ABB RobotStudio station: Yummi-Pick-and-Place.rsstn

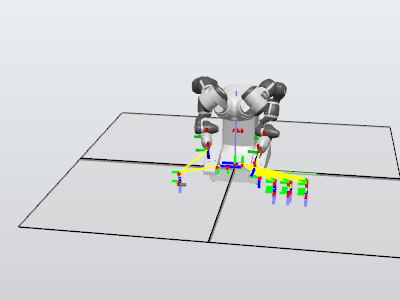
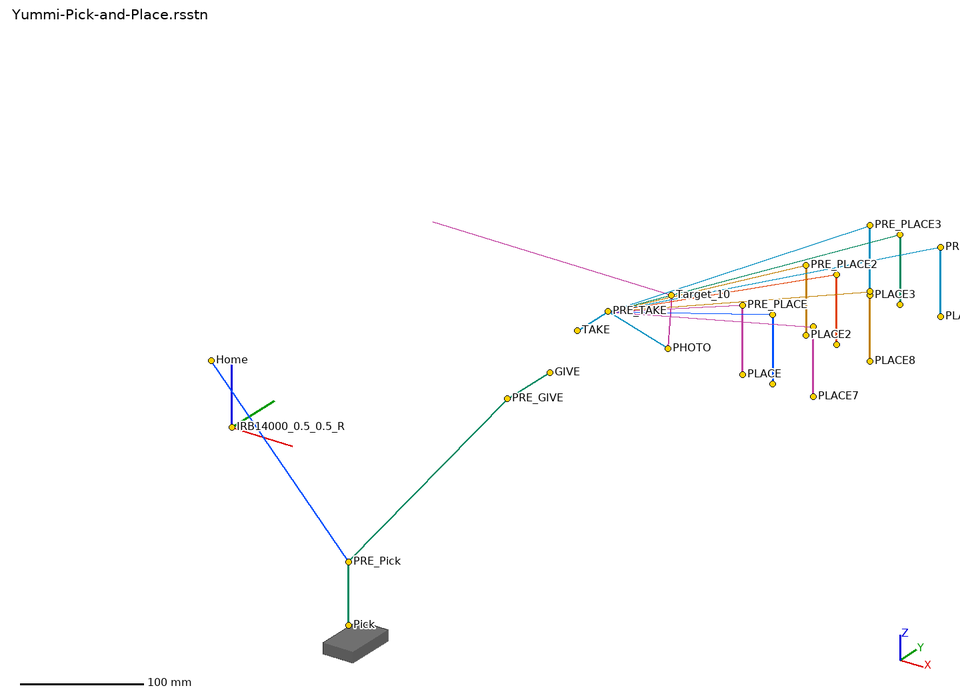
[picture v1: parts stored in the station drawn from their meshes, with robot base, taught points and paths (robot models come from the ABB library and are not in the file)]
Station Yummi5 (saved by RobotStudio 24.3.10958.1)
Controller Controller12
  mechanical unit ROB_R: IRB14000_0.5_0.5_R, 6 joints, base frame (0, 0, 0) mm
  mechanical unit ROB_R_7: IRB14000_0.5_0.5_R, 1 joints, base frame (0, 0, 0) mm
  mechanical unit ROB_L: IRB14000_0.5_0.5_L, 6 joints, base frame (0, 0, 0) mm
  mechanical unit ROB_L_7: IRB14000_0.5_0.5_L, 1 joints, base frame (0, 0, 0) mm
Layout (positions relative to the parent item):
  - IRB14000_0.5_0.5 [mechanism, from %ABB.RobotStudio.Models.IRB14000%\IRB14000_0.5_0.5__02.rslib] at (0, 0, 0) mm
  - IRB14000_0.5_0.5_R [mechanism, from %ABB.RobotStudio.Models.IRB14000%\IRB14000_0.5_0.5__02.rslib] at (0, 0, 0) mm; joint values [1.3686, -2.3546, -0.9667, 0.4669, -1.2245, 1.4931, 2.9439] (rad or m)
  - IRB14000_0.5_0.5_L [mechanism, from %ABB.RobotStudio.Models.IRB14000%\IRB14000_0.5_0.5__02.rslib] at (0, 0, 0) mm; joint values [-1.4023, -1.9659, 0.2989, 0.1537, 2.388, 1.6864, -2.7781] (rad or m)
  - Smart_Gripper_Servo_Fingers [mechanism] at (-9.58, -182.61, 198.63) mm, rotated rx 179.34 ry -63.63 rz 15.45 deg; joint values [0.02] (rad or m)
      TCP Servo at (0, 0, 114.2) mm
      links: HandBase, DownFinger, UpFinger, VacuumOne, VacuumTwo
  - Smart_Gripper_Servo_Fingers_2 [mechanism] at (-9.58, 182.61, 198.63) mm, rotated rx -179.34 ry -63.63 rz -15.45 deg; joint values [0.02] (rad or m)
      TCP Servo at (0, 0, 114.2) mm
      links: HandBase, DownFinger, UpFinger, VacuumOne, VacuumTwo
  - Part_2 [part] at (100, 0, 0) mm, size 30 x 50 x 10 mm
  - Part_3 [part], size 30 x 50 x 10 mm
  - Part_4 [part], size 30 x 50 x 10 mm
  - Part_5 [part], size 30 x 50 x 10 mm
  - Part_6 [part], size 30 x 50 x 10 mm
  - Part_7 [part], size 30 x 50 x 10 mm
  - Part_8 [part], size 30 x 50 x 10 mm
  - Part_9 [part], size 30 x 50 x 10 mm
  - Part_10 [part], size 30 x 50 x 10 mm
Attachment: Smart_Gripper_Servo_Fingers is attached to IRB14000_0.5_0.5_R / Link7
Attachment: Smart_Gripper_Servo_Fingers_2 is attached to IRB14000_0.5_0.5_L / Link7
EventTableEntry 3683: Group=, Trigger=GripperR 3684, Actions=[EventTableActionMechanicalPose 4791, EventTableActionAttach 4792], Comment=, ActivationMode=2, Cyclic=false
EventTableTriggerIO 3684: IOValue=[1], IRC5Controller=? -1, Operator=0, SignalSource=Controller12 1195
EventTableTriggerIO 3686: IOValue=[0], IRC5Controller=? -1, Operator=0, SignalSource=Controller12 1195
EventTableTriggerIO 3687: IOValue=[1], IRC5Controller=? -1, Operator=0, SignalSource=Controller12 1195
EventTableTriggerIO 3688: IOValue=[0], IRC5Controller=? -1, Operator=0, SignalSource=Controller12 1195
EventTableTriggerIO 3689: IOValue=[1], IRC5Controller=? -1, Operator=0, SignalSource=Controller12 1195
EventTableTriggerIO 3690: IOValue=[0], IRC5Controller=? -1, Operator=0, SignalSource=Controller12 1195
EventTableTriggerIO 3691: IOValue=[1], IRC5Controller=? -1, Operator=0, SignalSource=Controller12 1195
EventTableTriggerIO 3692: IOValue=[0], IRC5Controller=? -1, Operator=0, SignalSource=Controller12 1195
EventTableTriggerIO 3693: IOValue=[1], IRC5Controller=? -1, Operator=0, SignalSource=Controller12 1195
EventTableTriggerIO 3694: IOValue=[0], IRC5Controller=? -1, Operator=0, SignalSource=Controller12 1195
EventTableEntry 3695: Group=, Trigger=GripperR 3686, Actions=[EventTableActionMechanicalPose 3696, EventTableActionDetach 4527], Comment=, ActivationMode=2, Cyclic=false
EventTableActionMechanicalPose 3696: VirtualSignal=, Mechanism=Smart_Gripper_Servo_Fingers 3661, ToPoseName=Pose2, VirtualSignalValue=[1]
EventTableTriggerIO 3853: IOValue=[1], IRC5Controller=? -1, Operator=0, SignalSource=Controller12 1195
EventTableTriggerIO 3854: IOValue=[0], IRC5Controller=? -1, Operator=0, SignalSource=Controller12 1195
EventTableTriggerIO 3855: IOValue=[1], IRC5Controller=? -1, Operator=0, SignalSource=Controller12 1195
EventTableTriggerIO 3856: IOValue=[0], IRC5Controller=? -1, Operator=0, SignalSource=Controller12 1195
EventTableEntry 4149: Group=, Trigger=GripperL 4150, Actions=[EventTableActionMechanicalPose 4151, EventTableActionAttach 4528], Comment=, ActivationMode=2, Cyclic=false
EventTableTriggerIO 4150: IOValue=[1], IRC5Controller=? -1, Operator=0, SignalSource=Controller12 1195
EventTableActionMechanicalPose 4151: VirtualSignal=, Mechanism=Smart_Gripper_Servo_Fingers_2 3668, ToPoseName=Pose1, VirtualSignalValue=[1]
EventTableTriggerIO 4152: IOValue=[0], IRC5Controller=? -1, Operator=0, SignalSource=Controller12 1195
EventTableEntry 4153: Group=, Trigger=GripperL 4152, Actions=[EventTableActionMechanicalPose 4154, EventTableActionDetach 4529], Comment=, ActivationMode=2, Cyclic=false
EventTableActionMechanicalPose 4154: VirtualSignal=, Mechanism=Smart_Gripper_Servo_Fingers_2 3668, ToPoseName=Pose2, VirtualSignalValue=[1]
EventTableTriggerIO 4291: IOValue=[1], IRC5Controller=? -1, Operator=0, SignalSource=Controller12 1195
EventTableTriggerIO 4292: IOValue=[0], IRC5Controller=? -1, Operator=0, SignalSource=Controller12 1195
EventTableTriggerIO 4293: IOValue=[1], IRC5Controller=? -1, Operator=0, SignalSource=Controller12 1195
EventTableTriggerIO 4294: IOValue=[0], IRC5Controller=? -1, Operator=0, SignalSource=Controller12 1195
EventTableActionDetach 4527: AttachmentParent=Smart_Gripper_Servo_Fingers 3661, AttachmentChild=Part_2 4525
EventTableActionAttach 4528: AttachmentParent=Smart_Gripper_Servo_Fingers_2 3668, AttachmentChild=Part_2 4525, MountObject=false, Offset=[X=1, Y=0, Z=0, W=0, X=0, Y=1, Z=0, W=0, X=0, Y=0, Z=1, W=0, X=0, Y=0, Z=0, W=1], FlangeIndext=0, FindNearest=false
EventTableActionDetach 4529: AttachmentParent=Smart_Gripper_Servo_Fingers_2 3668, AttachmentChild=Part_2 4525
EventTableActionMechanicalPose 4791: VirtualSignal=, Mechanism=Smart_Gripper_Servo_Fingers 3661, ToPoseName=Pose1, VirtualSignalValue=[1]
EventTableActionAttach 4792: AttachmentParent=Smart_Gripper_Servo_Fingers 3661, AttachmentChild=Part_2 4525, MountObject=false, Offset=[X=1, Y=0, Z=0, W=0, X=0, Y=1, Z=0, W=0, X=0, Y=0, Z=1, W=0, X=0, Y=0, Z=0, W=1], FlangeIndext=0, FindNearest=false
EventTableEntry 6433: Group=, Trigger=GripperR_9 6434, Actions=[EventTableActionMechanicalPose 6435, EventTableActionAttach 6437], Comment=, ActivationMode=2, Cyclic=false
EventTableTriggerIO 6434: IOValue=[1], IRC5Controller=? -1, Operator=0, SignalSource=Controller12 1195
EventTableActionMechanicalPose 6435: VirtualSignal=, Mechanism=Smart_Gripper_Servo_Fingers 3661, ToPoseName=Pose1, VirtualSignalValue=[1]
EventTableTriggerIO 6436: IOValue=[0], IRC5Controller=? -1, Operator=0, SignalSource=Controller12 1195
EventTableActionAttach 6437: AttachmentParent=Smart_Gripper_Servo_Fingers 3661, AttachmentChild=Part_9 6430, MountObject=false, Offset=[X=1, Y=0, Z=0, W=0, X=0, Y=1, Z=0, W=0, X=0, Y=0, Z=1, W=0, X=0, Y=0, Z=0, W=1], FlangeIndext=0, FindNearest=false
EventTableEntry 6438: Group=, Trigger=GripperR_3 6439, Actions=[EventTableActionMechanicalPose 6440, EventTableActionAttach 6442], Comment=, ActivationMode=2, Cyclic=false
EventTableTriggerIO 6439: IOValue=[1], IRC5Controller=? -1, Operator=0, SignalSource=Controller12 1195
EventTableActionMechanicalPose 6440: VirtualSignal=, Mechanism=Smart_Gripper_Servo_Fingers 3661, ToPoseName=Pose1, VirtualSignalValue=[1]
EventTableTriggerIO 6441: IOValue=[0], IRC5Controller=? -1, Operator=0, SignalSource=Controller12 1195
EventTableActionAttach 6442: AttachmentParent=Smart_Gripper_Servo_Fingers 3661, AttachmentChild=Part_3 6418, MountObject=false, Offset=[X=1, Y=0, Z=0, W=0, X=0, Y=1, Z=0, W=0, X=0, Y=0, Z=1, W=0, X=0, Y=0, Z=0, W=1], FlangeIndext=0, FindNearest=false
EventTableEntry 6443: Group=, Trigger=GripperR_4 6444, Actions=[EventTableActionMechanicalPose 6445, EventTableActionAttach 6447], Comment=, ActivationMode=2, Cyclic=false
EventTableTriggerIO 6444: IOValue=[1], IRC5Controller=? -1, Operator=0, SignalSource=Controller12 1195
EventTableActionMechanicalPose 6445: VirtualSignal=, Mechanism=Smart_Gripper_Servo_Fingers 3661, ToPoseName=Pose1, VirtualSignalValue=[1]
EventTableTriggerIO 6446: IOValue=[0], IRC5Controller=? -1, Operator=0, SignalSource=Controller12 1195
EventTableActionAttach 6447: AttachmentParent=Smart_Gripper_Servo_Fingers 3661, AttachmentChild=Part_4 6420, MountObject=false, Offset=[X=1, Y=0, Z=0, W=0, X=0, Y=1, Z=0, W=0, X=0, Y=0, Z=1, W=0, X=0, Y=0, Z=0, W=1], FlangeIndext=0, FindNearest=false
EventTableEntry 6448: Group=, Trigger=GripperR_5 6449, Actions=[EventTableActionMechanicalPose 6450, EventTableActionAttach 6452], Comment=, ActivationMode=2, Cyclic=false
EventTableTriggerIO 6449: IOValue=[1], IRC5Controller=? -1, Operator=0, SignalSource=Controller12 1195
EventTableActionMechanicalPose 6450: VirtualSignal=, Mechanism=Smart_Gripper_Servo_Fingers 3661, ToPoseName=Pose1, VirtualSignalValue=[1]
EventTableTriggerIO 6451: IOValue=[0], IRC5Controller=? -1, Operator=0, SignalSource=Controller12 1195
EventTableActionAttach 6452: AttachmentParent=Smart_Gripper_Servo_Fingers 3661, AttachmentChild=Part_5 6422, MountObject=false, Offset=[X=1, Y=0, Z=0, W=0, X=0, Y=1, Z=0, W=0, X=0, Y=0, Z=1, W=0, X=0, Y=0, Z=0, W=1], FlangeIndext=0, FindNearest=false
EventTableEntry 6453: Group=, Trigger=GripperR_6 6454, Actions=[EventTableActionMechanicalPose 6455, EventTableActionAttach 6457], Comment=, ActivationMode=2, Cyclic=false
EventTableTriggerIO 6454: IOValue=[1], IRC5Controller=? -1, Operator=0, SignalSource=Controller12 1195
EventTableActionMechanicalPose 6455: VirtualSignal=, Mechanism=Smart_Gripper_Servo_Fingers 3661, ToPoseName=Pose1, VirtualSignalValue=[1]
EventTableTriggerIO 6456: IOValue=[0], IRC5Controller=? -1, Operator=0, SignalSource=Controller12 1195
EventTableActionAttach 6457: AttachmentParent=Smart_Gripper_Servo_Fingers 3661, AttachmentChild=Part_6 6424, MountObject=false, Offset=[X=1, Y=0, Z=0, W=0, X=0, Y=1, Z=0, W=0, X=0, Y=0, Z=1, W=0, X=0, Y=0, Z=0, W=1], FlangeIndext=0, FindNearest=false
EventTableEntry 6458: Group=, Trigger=GripperR_7 6459, Actions=[EventTableActionMechanicalPose 6460, EventTableActionAttach 6462], Comment=, ActivationMode=2, Cyclic=false
EventTableTriggerIO 6459: IOValue=[1], IRC5Controller=? -1, Operator=0, SignalSource=Controller12 1195
EventTableActionMechanicalPose 6460: VirtualSignal=, Mechanism=Smart_Gripper_Servo_Fingers 3661, ToPoseName=Pose1, VirtualSignalValue=[1]
EventTableTriggerIO 6461: IOValue=[0], IRC5Controller=? -1, Operator=0, SignalSource=Controller12 1195
EventTableActionAttach 6462: AttachmentParent=Smart_Gripper_Servo_Fingers 3661, AttachmentChild=Part_7 6426, MountObject=false, Offset=[X=1, Y=0, Z=0, W=0, X=0, Y=1, Z=0, W=0, X=0, Y=0, Z=1, W=0, X=0, Y=0, Z=0, W=1], FlangeIndext=0, FindNearest=false
EventTableEntry 6463: Group=, Trigger=GripperR_8 6464, Actions=[EventTableActionMechanicalPose 6465, EventTableActionAttach 6467], Comment=, ActivationMode=2, Cyclic=false
EventTableTriggerIO 6464: IOValue=[1], IRC5Controller=? -1, Operator=0, SignalSource=Controller12 1195
EventTableActionMechanicalPose 6465: VirtualSignal=, Mechanism=Smart_Gripper_Servo_Fingers 3661, ToPoseName=Pose1, VirtualSignalValue=[1]
EventTableTriggerIO 6466: IOValue=[0], IRC5Controller=? -1, Operator=0, SignalSource=Controller12 1195
EventTableActionAttach 6467: AttachmentParent=Smart_Gripper_Servo_Fingers 3661, AttachmentChild=Part_8 6428, MountObject=false, Offset=[X=1, Y=0, Z=0, W=0, X=0, Y=1, Z=0, W=0, X=0, Y=0, Z=1, W=0, X=0, Y=0, Z=0, W=1], FlangeIndext=0, FindNearest=false
EventTableEntry 6468: Group=, Trigger=GripperR_10 6469, Actions=[EventTableActionMechanicalPose 6470, EventTableActionAttach 6472], Comment=, ActivationMode=2, Cyclic=false
EventTableTriggerIO 6469: IOValue=[1], IRC5Controller=? -1, Operator=0, SignalSource=Controller12 1195
EventTableActionMechanicalPose 6470: VirtualSignal=, Mechanism=Smart_Gripper_Servo_Fingers 3661, ToPoseName=Pose1, VirtualSignalValue=[1]
EventTableTriggerIO 6471: IOValue=[0], IRC5Controller=? -1, Operator=0, SignalSource=Controller12 1195
EventTableActionAttach 6472: AttachmentParent=Smart_Gripper_Servo_Fingers 3661, AttachmentChild=Part_10 6432, MountObject=false, Offset=[X=1, Y=0, Z=0, W=0, X=0, Y=1, Z=0, W=0, X=0, Y=0, Z=1, W=0, X=0, Y=0, Z=0, W=1], FlangeIndext=0, FindNearest=false
EventTableEntry 6473: Group=, Trigger=GripperL_3 6474, Actions=[EventTableActionMechanicalPose 6475, EventTableActionAttach 6477], Comment=, ActivationMode=2, Cyclic=false
EventTableTriggerIO 6474: IOValue=[1], IRC5Controller=? -1, Operator=0, SignalSource=Controller12 1195
EventTableActionMechanicalPose 6475: VirtualSignal=, Mechanism=Smart_Gripper_Servo_Fingers_2 3668, ToPoseName=Pose1, VirtualSignalValue=[1]
EventTableTriggerIO 6476: IOValue=[0], IRC5Controller=? -1, Operator=0, SignalSource=Controller12 1195
EventTableActionAttach 6477: AttachmentParent=Smart_Gripper_Servo_Fingers_2 3668, AttachmentChild=Part_3 6418, MountObject=false, Offset=[X=1, Y=0, Z=0, W=0, X=0, Y=1, Z=0, W=0, X=0, Y=0, Z=1, W=0, X=0, Y=0, Z=0, W=1], FlangeIndext=0, FindNearest=false
EventTableEntry 6478: Group=, Trigger=GripperL_4 6479, Actions=[EventTableActionMechanicalPose 6480, EventTableActionAttach 6482], Comment=, ActivationMode=2, Cyclic=false
EventTableTriggerIO 6479: IOValue=[1], IRC5Controller=? -1, Operator=0, SignalSource=Controller12 1195
EventTableActionMechanicalPose 6480: VirtualSignal=, Mechanism=Smart_Gripper_Servo_Fingers_2 3668, ToPoseName=Pose1, VirtualSignalValue=[1]
EventTableTriggerIO 6481: IOValue=[0], IRC5Controller=? -1, Operator=0, SignalSource=Controller12 1195
EventTableActionAttach 6482: AttachmentParent=Smart_Gripper_Servo_Fingers_2 3668, AttachmentChild=Part_4 6420, MountObject=false, Offset=[X=1, Y=0, Z=0, W=0, X=0, Y=1, Z=0, W=0, X=0, Y=0, Z=1, W=0, X=0, Y=0, Z=0, W=1], FlangeIndext=0, FindNearest=false
EventTableEntry 6483: Group=, Trigger=GripperL_5 6484, Actions=[EventTableActionMechanicalPose 6485, EventTableActionAttach 6487], Comment=, ActivationMode=2, Cyclic=false
EventTableTriggerIO 6484: IOValue=[1], IRC5Controller=? -1, Operator=0, SignalSource=Controller12 1195
EventTableActionMechanicalPose 6485: VirtualSignal=, Mechanism=Smart_Gripper_Servo_Fingers_2 3668, ToPoseName=Pose1, VirtualSignalValue=[1]
EventTableTriggerIO 6486: IOValue=[0], IRC5Controller=? -1, Operator=0, SignalSource=Controller12 1195
EventTableActionAttach 6487: AttachmentParent=Smart_Gripper_Servo_Fingers_2 3668, AttachmentChild=Part_5 6422, MountObject=false, Offset=[X=1, Y=0, Z=0, W=0, X=0, Y=1, Z=0, W=0, X=0, Y=0, Z=1, W=0, X=0, Y=0, Z=0, W=1], FlangeIndext=0, FindNearest=false
EventTableEntry 6488: Group=, Trigger=GripperL_6 6489, Actions=[EventTableActionMechanicalPose 6490, EventTableActionAttach 6492], Comment=, ActivationMode=2, Cyclic=false
EventTableTriggerIO 6489: IOValue=[1], IRC5Controller=? -1, Operator=0, SignalSource=Controller12 1195
EventTableActionMechanicalPose 6490: VirtualSignal=, Mechanism=Smart_Gripper_Servo_Fingers_2 3668, ToPoseName=Pose1, VirtualSignalValue=[1]
EventTableTriggerIO 6491: IOValue=[0], IRC5Controller=? -1, Operator=0, SignalSource=Controller12 1195
EventTableActionAttach 6492: AttachmentParent=Smart_Gripper_Servo_Fingers_2 3668, AttachmentChild=Part_6 6424, MountObject=false, Offset=[X=1, Y=0, Z=0, W=0, X=0, Y=1, Z=0, W=0, X=0, Y=0, Z=1, W=0, X=0, Y=0, Z=0, W=1], FlangeIndext=0, FindNearest=false
EventTableEntry 6493: Group=, Trigger=GripperL_7 6494, Actions=[EventTableActionMechanicalPose 6495, EventTableActionAttach 6497], Comment=, ActivationMode=2, Cyclic=false
EventTableTriggerIO 6494: IOValue=[1], IRC5Controller=? -1, Operator=0, SignalSource=Controller12 1195
EventTableActionMechanicalPose 6495: VirtualSignal=, Mechanism=Smart_Gripper_Servo_Fingers_2 3668, ToPoseName=Pose1, VirtualSignalValue=[1]
EventTableTriggerIO 6496: IOValue=[0], IRC5Controller=? -1, Operator=0, SignalSource=Controller12 1195
EventTableActionAttach 6497: AttachmentParent=Smart_Gripper_Servo_Fingers_2 3668, AttachmentChild=Part_7 6426, MountObject=false, Offset=[X=1, Y=0, Z=0, W=0, X=0, Y=1, Z=0, W=0, X=0, Y=0, Z=1, W=0, X=0, Y=0, Z=0, W=1], FlangeIndext=0, FindNearest=false
EventTableEntry 6498: Group=, Trigger=GripperL_8 6499, Actions=[EventTableActionMechanicalPose 6500, EventTableActionAttach 6547], Comment=, ActivationMode=2, Cyclic=false
EventTableTriggerIO 6499: IOValue=[1], IRC5Controller=? -1, Operator=0, SignalSource=Controller12 1195
EventTableActionMechanicalPose 6500: VirtualSignal=, Mechanism=Smart_Gripper_Servo_Fingers_2 3668, ToPoseName=Pose1, VirtualSignalValue=[1]
EventTableEntry 6501: Group=, Trigger=GripperL_9 6502, Actions=[EventTableActionMechanicalPose 6503, EventTableActionAttach 6549], Comment=, ActivationMode=2, Cyclic=false
EventTableTriggerIO 6502: IOValue=[1], IRC5Controller=? -1, Operator=0, SignalSource=Controller12 1195
EventTableActionMechanicalPose 6503: VirtualSignal=, Mechanism=Smart_Gripper_Servo_Fingers_2 3668, ToPoseName=Pose1, VirtualSignalValue=[1]
EventTableEntry 6504: Group=, Trigger=GripperL_10 6505, Actions=[EventTableActionMechanicalPose 6506, EventTableActionAttach 6551], Comment=, ActivationMode=2, Cyclic=false
EventTableTriggerIO 6505: IOValue=[1], IRC5Controller=? -1, Operator=0, SignalSource=Controller12 1195
EventTableActionMechanicalPose 6506: VirtualSignal=, Mechanism=Smart_Gripper_Servo_Fingers_2 3668, ToPoseName=Pose1, VirtualSignalValue=[1]
EventTableEntry 6507: Group=, Trigger=GripperR_9 6436, Actions=[EventTableActionMechanicalPose 6508, EventTableActionDetach 6509], Comment=, ActivationMode=2, Cyclic=false
EventTableActionMechanicalPose 6508: VirtualSignal=, Mechanism=Smart_Gripper_Servo_Fingers 3661, ToPoseName=Pose2, VirtualSignalValue=[1]
EventTableActionDetach 6509: AttachmentParent=Smart_Gripper_Servo_Fingers 3661, AttachmentChild=Part_9 6430
EventTableEntry 6510: Group=, Trigger=GripperR_3 6441, Actions=[EventTableActionMechanicalPose 6511, EventTableActionDetach 6512], Comment=, ActivationMode=2, Cyclic=false
EventTableActionMechanicalPose 6511: VirtualSignal=, Mechanism=Smart_Gripper_Servo_Fingers 3661, ToPoseName=Pose2, VirtualSignalValue=[1]
EventTableActionDetach 6512: AttachmentParent=Smart_Gripper_Servo_Fingers 3661, AttachmentChild=Part_3 6418
EventTableEntry 6513: Group=, Trigger=GripperR_4 6446, Actions=[EventTableActionMechanicalPose 6514, EventTableActionDetach 6515], Comment=, ActivationMode=2, Cyclic=false
EventTableActionMechanicalPose 6514: VirtualSignal=, Mechanism=Smart_Gripper_Servo_Fingers 3661, ToPoseName=Pose2, VirtualSignalValue=[1]
EventTableActionDetach 6515: AttachmentParent=Smart_Gripper_Servo_Fingers 3661, AttachmentChild=Part_4 6420
EventTableEntry 6516: Group=, Trigger=GripperR_5 6451, Actions=[EventTableActionMechanicalPose 6517, EventTableActionDetach 6518], Comment=, ActivationMode=2, Cyclic=false
EventTableActionMechanicalPose 6517: VirtualSignal=, Mechanism=Smart_Gripper_Servo_Fingers 3661, ToPoseName=Pose2, VirtualSignalValue=[1]
EventTableActionDetach 6518: AttachmentParent=Smart_Gripper_Servo_Fingers 3661, AttachmentChild=Part_5 6422
EventTableEntry 6519: Group=, Trigger=GripperR_6 6456, Actions=[EventTableActionMechanicalPose 6520, EventTableActionDetach 6521], Comment=, ActivationMode=2, Cyclic=false
EventTableActionMechanicalPose 6520: VirtualSignal=, Mechanism=Smart_Gripper_Servo_Fingers 3661, ToPoseName=Pose2, VirtualSignalValue=[1]
EventTableActionDetach 6521: AttachmentParent=Smart_Gripper_Servo_Fingers 3661, AttachmentChild=Part_6 6424
EventTableEntry 6522: Group=, Trigger=GripperR_7 6461, Actions=[EventTableActionMechanicalPose 6523, EventTableActionDetach 6524], Comment=, ActivationMode=2, Cyclic=false
EventTableActionMechanicalPose 6523: VirtualSignal=, Mechanism=Smart_Gripper_Servo_Fingers 3661, ToPoseName=Pose2, VirtualSignalValue=[1]
EventTableActionDetach 6524: AttachmentParent=Smart_Gripper_Servo_Fingers 3661, AttachmentChild=Part_7 6426
EventTableEntry 6525: Group=, Trigger=GripperR_8 6466, Actions=[EventTableActionMechanicalPose 6526, EventTableActionDetach 6527], Comment=, ActivationMode=2, Cyclic=false
EventTableActionMechanicalPose 6526: VirtualSignal=, Mechanism=Smart_Gripper_Servo_Fingers 3661, ToPoseName=Pose2, VirtualSignalValue=[1]
EventTableActionDetach 6527: AttachmentParent=Smart_Gripper_Servo_Fingers 3661, AttachmentChild=Part_8 6428
EventTableEntry 6528: Group=, Trigger=GripperR_10 6471, Actions=[EventTableActionMechanicalPose 6529, EventTableActionDetach 6530], Comment=, ActivationMode=2, Cyclic=false
EventTableActionMechanicalPose 6529: VirtualSignal=, Mechanism=Smart_Gripper_Servo_Fingers 3661, ToPoseName=Pose2, VirtualSignalValue=[1]
EventTableActionDetach 6530: AttachmentParent=Smart_Gripper_Servo_Fingers 3661, AttachmentChild=Part_10 6432
EventTableEntry 6531: Group=, Trigger=GripperL_3 6476, Actions=[EventTableActionMechanicalPose 6532, EventTableActionDetach 6533], Comment=, ActivationMode=2, Cyclic=false
EventTableActionMechanicalPose 6532: VirtualSignal=, Mechanism=Smart_Gripper_Servo_Fingers_2 3668, ToPoseName=Pose2, VirtualSignalValue=[1]
EventTableActionDetach 6533: AttachmentParent=Smart_Gripper_Servo_Fingers_2 3668, AttachmentChild=Part_3 6418
EventTableEntry 6534: Group=, Trigger=GripperL_4 6481, Actions=[EventTableActionMechanicalPose 6535, EventTableActionDetach 6536], Comment=, ActivationMode=2, Cyclic=false
EventTableActionMechanicalPose 6535: VirtualSignal=, Mechanism=Smart_Gripper_Servo_Fingers_2 3668, ToPoseName=Pose2, VirtualSignalValue=[1]
EventTableActionDetach 6536: AttachmentParent=Smart_Gripper_Servo_Fingers_2 3668, AttachmentChild=Part_4 6420
EventTableEntry 6537: Group=, Trigger=GripperL_5 6486, Actions=[EventTableActionMechanicalPose 6538, EventTableActionDetach 6539], Comment=, ActivationMode=2, Cyclic=false
EventTableActionMechanicalPose 6538: VirtualSignal=, Mechanism=Smart_Gripper_Servo_Fingers_2 3668, ToPoseName=Pose2, VirtualSignalValue=[1]
EventTableActionDetach 6539: AttachmentParent=Smart_Gripper_Servo_Fingers_2 3668, AttachmentChild=Part_5 6422
EventTableEntry 6540: Group=, Trigger=GripperL_6 6491, Actions=[EventTableActionMechanicalPose 6541, EventTableActionDetach 6542], Comment=, ActivationMode=2, Cyclic=false
EventTableActionMechanicalPose 6541: VirtualSignal=, Mechanism=Smart_Gripper_Servo_Fingers_2 3668, ToPoseName=Pose2, VirtualSignalValue=[1]
EventTableActionDetach 6542: AttachmentParent=Smart_Gripper_Servo_Fingers_2 3668, AttachmentChild=Part_6 6424
EventTableEntry 6543: Group=, Trigger=GripperL_7 6496, Actions=[EventTableActionMechanicalPose 6544, EventTableActionDetach 6545], Comment=, ActivationMode=2, Cyclic=false
EventTableActionMechanicalPose 6544: VirtualSignal=, Mechanism=Smart_Gripper_Servo_Fingers_2 3668, ToPoseName=Pose2, VirtualSignalValue=[1]
EventTableActionDetach 6545: AttachmentParent=Smart_Gripper_Servo_Fingers_2 3668, AttachmentChild=Part_7 6426
EventTableTriggerIO 6546: IOValue=[0], IRC5Controller=? -1, Operator=0, SignalSource=Controller12 1195
EventTableActionAttach 6547: AttachmentParent=Smart_Gripper_Servo_Fingers_2 3668, AttachmentChild=Part_8 6428, MountObject=true, Offset=[X=1, Y=0, Z=0, W=0, X=0, Y=1, Z=0, W=0, X=0, Y=0, Z=1, W=0, X=0, Y=0, Z=0, W=1], FlangeIndext=0, FindNearest=false
EventTableTriggerIO 6548: IOValue=[0], IRC5Controller=? -1, Operator=0, SignalSource=Controller12 1195
EventTableActionAttach 6549: AttachmentParent=Smart_Gripper_Servo_Fingers_2 3668, AttachmentChild=Part_9 6430, MountObject=false, Offset=[X=1, Y=0, Z=0, W=0, X=0, Y=1, Z=0, W=0, X=0, Y=0, Z=1, W=0, X=0, Y=0, Z=0, W=1], FlangeIndext=0, FindNearest=false
EventTableTriggerIO 6550: IOValue=[0], IRC5Controller=? -1, Operator=0, SignalSource=Controller12 1195
EventTableActionAttach 6551: AttachmentParent=Smart_Gripper_Servo_Fingers_2 3668, AttachmentChild=Part_10 6432, MountObject=false, Offset=[X=1, Y=0, Z=0, W=0, X=0, Y=1, Z=0, W=0, X=0, Y=0, Z=1, W=0, X=0, Y=0, Z=0, W=1], FlangeIndext=0, FindNearest=false
EventTableEntry 6552: Group=, Trigger=GripperL_8 6546, Actions=[EventTableActionMechanicalPose 6553, EventTableActionDetach 6554], Comment=, ActivationMode=2, Cyclic=false
EventTableActionMechanicalPose 6553: VirtualSignal=, Mechanism=Smart_Gripper_Servo_Fingers_2 3668, ToPoseName=Pose2, VirtualSignalValue=[1]
EventTableActionDetach 6554: AttachmentParent=Smart_Gripper_Servo_Fingers_2 3668, AttachmentChild=Part_8 6428
EventTableEntry 6555: Group=, Trigger=GripperL_9 6548, Actions=[EventTableActionMechanicalPose 6556, EventTableActionDetach 6557], Comment=, ActivationMode=2, Cyclic=false
EventTableActionMechanicalPose 6556: VirtualSignal=, Mechanism=Smart_Gripper_Servo_Fingers_2 3668, ToPoseName=Pose2, VirtualSignalValue=[1]
EventTableActionDetach 6557: AttachmentParent=Smart_Gripper_Servo_Fingers_2 3668, AttachmentChild=Part_9 6430
EventTableEntry 6558: Group=, Trigger=GripperL_10 6550, Actions=[EventTableActionMechanicalPose 6559, EventTableActionDetach 6560], Comment=, ActivationMode=2, Cyclic=false
EventTableActionMechanicalPose 6559: VirtualSignal=, Mechanism=Smart_Gripper_Servo_Fingers_2 3668, ToPoseName=Pose2, VirtualSignalValue=[1]
EventTableActionDetach 6560: AttachmentParent=Smart_Gripper_Servo_Fingers_2 3668, AttachmentChild=Part_10 6432
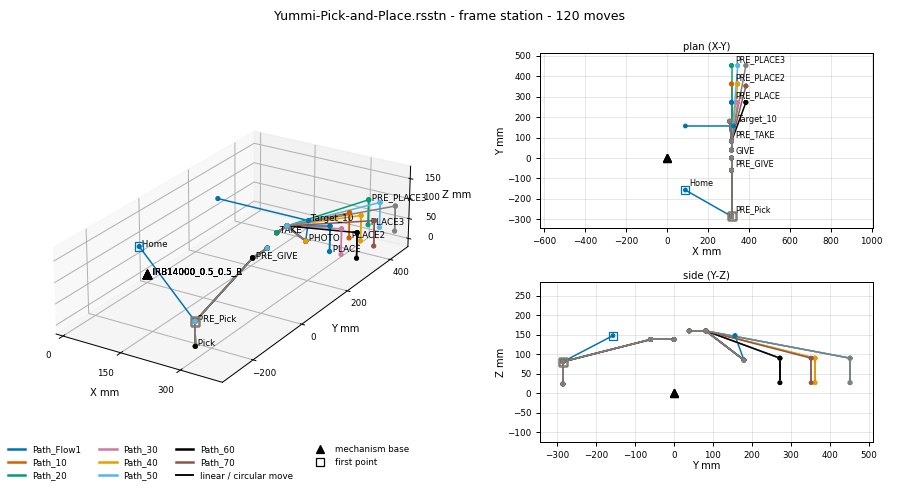
[picture p0: tool path of Yummi-Pick-and-Place.rsstn in frame station, 120 of 120 moves have a stored position in this frame; points joined in program order, loops and branches not executed]
Targets, tools, work objects and paths stored in the station, written as RAPID:
! task T_ROB_R
MODULE CalibData
  PERS tooldata Servo:=[TRUE,[[0,0,114.2],[1,0,0,0]],[0.215,[8.7,12.3,49.2],[1,0,0,0],0.00021,0.00024,0.00009]];
ENDMODULE

! task T_ROB_R
MODULE Module1
  CONST robtarget Pick:=[[315,-285,23.743],[0,1,0,0],[1,-2,2,4],[-106.008706385,9E+09,9E+09,9E+09,9E+09,9E+09]];
  CONST robtarget Home:=[[89.387946422,-156.622117956,147.913470217],[0.066010726,-0.842420918,-0.111214912,-0.523068661],[0,0,0,4],[-101.964427132,9E+09,9E+09,9E+09,9E+09,9E+09]];
  CONST robtarget PRE_Pick:=[[315,-285.001,80.881],[0,1,0,0],[0,-2,2,4],[-106.008708916,9E+09,9E+09,9E+09,9E+09,9E+09]];
  CONST robtarget GIVE:=[[315,0,138],[0.707106781,-0.707106781,0,0],[1,-1,2,4],[-106.008705488,9E+09,9E+09,9E+09,9E+09,9E+09]];
  CONST robtarget PRE_GIVE:=[[315,-60,138],[0.707106781,-0.707106781,0,0],[1,-1,2,4],[-106.008709879,9E+09,9E+09,9E+09,9E+09,9E+09]];
  PROC main()
    Path_Flow1;
    Path_10;
    Path_20;
    Path_30;
    Path_40;
    Path_50;
    Path_60;
    Path_70;
    Path_80;
  ENDPROC
  PROC Path_Flow1()
    MoveJ Home,v200,fine,Servo\WObj:=wobj0;
    MoveL PRE_Pick,v200,z100,Servo\WObj:=wobj0;
    MoveL Pick,v200,z100,Servo\WObj:=wobj0;
    WaitTime 0.7;
    Set GripperR;
    MoveL PRE_Pick,v200,z100,Servo\WObj:=wobj0;
    MoveL PRE_GIVE,v200,z100,Servo\WObj:=wobj0;
    MoveL GIVE,v200,z100,Servo\WObj:=wobj0;
    WaitTime 0.5;
    Reset GripperR;
    MoveL PRE_GIVE,v200,z100,Servo\WObj:=wobj0;
  ENDPROC
  PROC Path_10()
    MoveL PRE_Pick,v200,z50,Servo\WObj:=wobj0;
    MoveL Pick,v200,z50,Servo\WObj:=wobj0;
    WaitTime 0.7;
    Set GripperR_3;
    MoveL PRE_Pick,v200,z50,Servo\WObj:=wobj0;
    MoveL PRE_GIVE,v200,z50,Servo\WObj:=wobj0;
    MoveL GIVE,v200,z50,Servo\WObj:=wobj0;
    WaitTime 0.5;
    Reset GripperR_3;
    MoveL PRE_GIVE,v200,z50,Servo\WObj:=wobj0;
  ENDPROC
  PROC Path_20()
    MoveL PRE_Pick,v200,z50,Servo\WObj:=wobj0;
    MoveL Pick,v200,z50,Servo\WObj:=wobj0;
    WaitTime 0.7;
    Set GripperR_4;
    MoveL PRE_Pick,v200,z50,Servo\WObj:=wobj0;
    MoveL PRE_GIVE,v200,z50,Servo\WObj:=wobj0;
    MoveL GIVE,v200,z50,Servo\WObj:=wobj0;
    WaitTime 0.5;
    Reset GripperR_4;
    MoveL PRE_GIVE,v200,z50,Servo\WObj:=wobj0;
  ENDPROC
  PROC Path_30()
    MoveL PRE_Pick,v200,z50,Servo\WObj:=wobj0;
    MoveL Pick,v200,z50,Servo\WObj:=wobj0;
    WaitTime 0.7;
    Set GripperR_5;
    MoveL PRE_Pick,v200,z50,Servo\WObj:=wobj0;
    MoveL PRE_GIVE,v200,z50,Servo\WObj:=wobj0;
    MoveL GIVE,v200,z50,Servo\WObj:=wobj0;
    WaitTime 0.5;
    Reset GripperR_5;
    MoveL PRE_GIVE,v200,z50,Servo\WObj:=wobj0;
  ENDPROC
  PROC Path_40()
    MoveL PRE_Pick,v200,z50,Servo\WObj:=wobj0;
    MoveL Pick,v200,z50,Servo\WObj:=wobj0;
    WaitTime 0.7;
    Set GripperR_6;
    MoveL PRE_Pick,v200,z50,Servo\WObj:=wobj0;
    MoveL PRE_GIVE,v200,z50,Servo\WObj:=wobj0;
    MoveL GIVE,v200,z50,Servo\WObj:=wobj0;
    WaitTime 0.5;
    Reset GripperR_6;
    MoveL PRE_GIVE,v200,z50,Servo\WObj:=wobj0;
  ENDPROC
  PROC Path_50()
    MoveL PRE_Pick,v200,z50,Servo\WObj:=wobj0;
    MoveL Pick,v200,z50,Servo\WObj:=wobj0;
    WaitTime 0.7;
    Set GripperR_7;
    MoveL PRE_Pick,v200,z50,Servo\WObj:=wobj0;
    MoveL PRE_GIVE,v200,z50,Servo\WObj:=wobj0;
    MoveL GIVE,v200,z50,Servo\WObj:=wobj0;
    WaitTime 0.5;
    Reset GripperR_7;
    MoveL PRE_GIVE,v200,z50,Servo\WObj:=wobj0;
  ENDPROC
  PROC Path_60()
    MoveL PRE_Pick,v200,z50,Servo\WObj:=wobj0;
    MoveL Pick,v200,z50,Servo\WObj:=wobj0;
    WaitTime 0.7;
    Set GripperR_8;
    MoveL PRE_Pick,v200,z50,Servo\WObj:=wobj0;
    MoveL PRE_GIVE,v200,z50,Servo\WObj:=wobj0;
    MoveL GIVE,v200,z50,Servo\WObj:=wobj0;
    WaitTime 0.5;
    Reset GripperR_8;
    MoveL PRE_GIVE,v200,z50,Servo\WObj:=wobj0;
  ENDPROC
  PROC Path_70()
    MoveL PRE_Pick,v200,z50,Servo\WObj:=wobj0;
    MoveL Pick,v200,z50,Servo\WObj:=wobj0;
    WaitTime 0.7;
    Set GripperR_9;
    MoveL PRE_Pick,v200,z50,Servo\WObj:=wobj0;
    MoveL PRE_GIVE,v200,z50,Servo\WObj:=wobj0;
    MoveL GIVE,v200,z50,Servo\WObj:=wobj0;
    WaitTime 0.5;
    Reset GripperR_9;
    MoveL PRE_GIVE,v200,z50,Servo\WObj:=wobj0;
  ENDPROC
  PROC Path_80()
    MoveL PRE_Pick,v200,z50,Servo\WObj:=wobj0;
    MoveL Pick,v200,z50,Servo\WObj:=wobj0;
    WaitTime 0.7;
    Set GripperR_10;
    MoveL PRE_Pick,v200,z50,Servo\WObj:=wobj0;
    MoveL PRE_GIVE,v200,z50,Servo\WObj:=wobj0;
    MoveL GIVE,v200,z50,Servo\WObj:=wobj0;
    WaitTime 0.5;
    Reset GripperR_10;
    MoveL PRE_GIVE,v200,z50,Servo\WObj:=wobj0;
  ENDPROC
ENDMODULE

! task T_ROB_L
MODULE CalibData
  PERS tooldata Servo:=[TRUE,[[0,0,114.2],[1,0,0,0]],[0.215,[8.7,12.3,49.2],[1,0,0,0],0.00021,0.00024,0.00009]];
ENDMODULE

! task T_ROB_L
MODULE Module1
  CONST robtarget Home:=[[89.387946423,156.622117957,147.913470217],[0.066010726,0.842420918,-0.111214912,0.523068661],[0,0,0,4],[101.964427132,9E+09,9E+09,9E+09,9E+09,9E+09]];
  CONST robtarget PRE_PHOTO:=[[305.763509464,179.639943254,85.193533141],[0.000218219,0.996549256,0.079302175,-0.02450915],[0,2,-2,4],[106.696431274,9E+09,9E+09,9E+09,9E+09,9E+09]];
  CONST robtarget PHOTO:=[[305.763594171,179.640203217,85.193485043],[0.000218113,0.996549254,0.079302152,-0.024509292],[-1,2,-2,4],[106.696427803,9E+09,9E+09,9E+09,9E+09,9E+09]];
  CONST robtarget TAKE:=[[315,39,160],[0.707106781,0.707106781,0,0],[-1,1,-2,4],[106.696423551,9E+09,9E+09,9E+09,9E+09,9E+09]];
  CONST robtarget PRE_TAKE:=[[315,82,160],[0.707106781,0.707106781,0,0],[-1,1,-2,4],[106.696423802,9E+09,9E+09,9E+09,9E+09,9E+09]];
  CONST robtarget PRE_PLACE:=[[315,272,90],[0,1,0,0],[-1,2,-2,4],[106.69642993,9E+09,9E+09,9E+09,9E+09,9E+09]];
  CONST robtarget PLACE:=[[315,272,27],[0,1,0,0],[-1,2,-2,4],[106.696421649,9E+09,9E+09,9E+09,9E+09,9E+09]];
  CONST robtarget Target_10:=[[325.684499399,156.622505768,147.913439612],[0.066010656,0.842421097,-0.111215044,0.523068353],[-1,2,-2,4],[106.780300148,9E+09,9E+09,9E+09,9E+09,9E+09]];
  CONST robtarget PRE_PLACE2:=[[315,362,90],[0,1,0,0],[-1,2,-2,4],[106.69642993,9E+09,9E+09,9E+09,9E+09,9E+09]];
  CONST robtarget PLACE2:=[[315,362,27],[0,1,0,0],[-1,2,-2,4],[106.696421649,9E+09,9E+09,9E+09,9E+09,9E+09]];
  CONST robtarget PRE_PLACE3:=[[315,452,90],[0,1,0,0],[-1,2,-2,4],[106.69642993,9E+09,9E+09,9E+09,9E+09,9E+09]];
  CONST robtarget PLACE3:=[[315,452,27],[0,1,0,0],[-1,2,-2,4],[106.696421649,9E+09,9E+09,9E+09,9E+09,9E+09]];
  CONST robtarget PRE_PLACE4:=[[345,272,90],[0,1,0,0],[-1,2,-2,4],[106.69642993,9E+09,9E+09,9E+09,9E+09,9E+09]];
  CONST robtarget PLACE4:=[[345,272,27],[0,1,0,0],[-1,2,-2,4],[106.696421649,9E+09,9E+09,9E+09,9E+09,9E+09]];
  CONST robtarget PRE_PLACE5:=[[345,362,90],[0,1,0,0],[-1,2,-2,4],[106.69642993,9E+09,9E+09,9E+09,9E+09,9E+09]];
  CONST robtarget PLACE5:=[[345,362,27],[0,1,0,0],[-1,2,-2,4],[106.696421649,9E+09,9E+09,9E+09,9E+09,9E+09]];
  CONST robtarget PRE_PLACE6:=[[345,452,90],[0,1,0,0],[-1,2,-2,4],[106.69642993,9E+09,9E+09,9E+09,9E+09,9E+09]];
  CONST robtarget PLACE6:=[[345,452,27],[0,1,0,0],[-1,2,-2,4],[106.696421649,9E+09,9E+09,9E+09,9E+09,9E+09]];
  CONST robtarget PRE_PLACE7:=[[385,272,90],[0,1,0,0],[-1,2,-2,4],[106.69642993,9E+09,9E+09,9E+09,9E+09,9E+09]];
  CONST robtarget PLACE7:=[[385,272,27],[0,1,0,0],[-1,2,-2,4],[106.696421649,9E+09,9E+09,9E+09,9E+09,9E+09]];
  CONST robtarget PRE_PLACE8:=[[385,352,90],[0,1,0,0],[-1,2,-2,4],[106.69642993,9E+09,9E+09,9E+09,9E+09,9E+09]];
  CONST robtarget PLACE8:=[[385,352,27],[0,1,0,0],[-1,2,-2,4],[106.696421649,9E+09,9E+09,9E+09,9E+09,9E+09]];
  CONST robtarget PRE_PLACE9:=[[385,452,90],[0,1,0,0],[-1,2,-2,4],[106.69642993,9E+09,9E+09,9E+09,9E+09,9E+09]];
  CONST robtarget PLACE9:=[[385,452,27],[0,1,0,0],[-1,2,-2,4],[106.696421649,9E+09,9E+09,9E+09,9E+09,9E+09]];
  PROC main()
    Path_Flow1;
    Path_10;
    Path_20;
    Path_30;
    Path_40;
    Path_50;
    Path_60;
    Path_70;
    Path_80;
  ENDPROC
  PROC Path_Flow1()
    MoveJ Home,v200,z100,Servo\WObj:=wobj0;
    MoveL Target_10,v200,z50,Servo\WObj:=wobj0;
    MoveL PHOTO,v200,z50,Servo\WObj:=wobj0;
    WaitTime 5;
    MoveL PRE_TAKE,v200,z50,Servo\WObj:=wobj0;
    MoveL TAKE,v200,z50,Servo\WObj:=wobj0;
    WaitTime 1;
    Set GripperL;
    WaitTime 1;
    MoveL PRE_TAKE,v200,z50,Servo\WObj:=wobj0;
    MoveL PRE_PLACE,v200,fine,Servo\WObj:=wobj0;
    MoveL PLACE,v200,fine,Servo\WObj:=wobj0;
    Reset GripperL;
    MoveL PRE_PLACE,v200,fine,Servo\WObj:=wobj0;
  ENDPROC
  PROC Path_10()
    MoveL PHOTO,v200,z50,Servo\WObj:=wobj0;
    WaitTime 5;
    MoveL PRE_TAKE,v200,z50,Servo\WObj:=wobj0;
    MoveL TAKE,v200,z50,Servo\WObj:=wobj0;
    WaitTime 1;
    Set GripperL_3;
    WaitTime 1;
    MoveL PRE_TAKE,v200,z50,Servo\WObj:=wobj0;
    MoveL PRE_PLACE2,v200,z50,Servo\WObj:=wobj0;
    MoveL PLACE2,v200,z50,Servo\WObj:=wobj0;
    Reset GripperL_3;
    MoveL PRE_PLACE2,v200,z50,Servo\WObj:=wobj0;
  ENDPROC
  PROC Path_20()
    MoveL PHOTO,v200,z50,Servo\WObj:=wobj0;
    WaitTime 5;
    MoveL PRE_TAKE,v200,z50,Servo\WObj:=wobj0;
    MoveL TAKE,v200,z50,Servo\WObj:=wobj0;
    WaitTime 1;
    Set GripperL_4;
    WaitTime 1;
    MoveL PRE_TAKE,v200,z50,Servo\WObj:=wobj0;
    MoveL PRE_PLACE3,v200,z50,Servo\WObj:=wobj0;
    MoveL PLACE3,v200,z50,Servo\WObj:=wobj0;
    Reset GripperL_4;
    MoveL PRE_PLACE3,v200,z50,Servo\WObj:=wobj0;
  ENDPROC
  PROC Path_30()
    MoveL PHOTO,v200,z50,Servo\WObj:=wobj0;
    WaitTime 5;
    MoveL PRE_TAKE,v200,z50,Servo\WObj:=wobj0;
    MoveL TAKE,v200,z50,Servo\WObj:=wobj0;
    WaitTime 1;
    Set GripperL_5;
    WaitTime 1;
    MoveL PRE_TAKE,v200,z50,Servo\WObj:=wobj0;
    MoveL PRE_PLACE4,v200,z50,Servo\WObj:=wobj0;
    MoveL PLACE4,v200,z50,Servo\WObj:=wobj0;
    Reset GripperL_5;
    MoveL PRE_PLACE4,v200,z50,Servo\WObj:=wobj0;
  ENDPROC
  PROC Path_40()
    MoveL PHOTO,v200,z50,Servo\WObj:=wobj0;
    WaitTime 5;
    MoveL PRE_TAKE,v200,z50,Servo\WObj:=wobj0;
    MoveL TAKE,v200,z50,Servo\WObj:=wobj0;
    WaitTime 1;
    Set GripperL_6;
    WaitTime 1;
    MoveL PRE_TAKE,v200,z50,Servo\WObj:=wobj0;
    MoveL PRE_PLACE5,v200,z50,Servo\WObj:=wobj0;
    MoveL PLACE5,v200,z50,Servo\WObj:=wobj0;
    Reset GripperL_6;
    MoveL PRE_PLACE5,v200,z50,Servo\WObj:=wobj0;
  ENDPROC
  PROC Path_50()
    MoveL PHOTO,v200,z50,Servo\WObj:=wobj0;
    WaitTime 5;
    MoveL PRE_TAKE,v200,z50,Servo\WObj:=wobj0;
    MoveL TAKE,v200,z50,Servo\WObj:=wobj0;
    WaitTime 1;
    Set GripperL_7;
    WaitTime 1;
    MoveL PRE_TAKE,v200,z50,Servo\WObj:=wobj0;
    MoveL PRE_PLACE6,v200,z50,Servo\WObj:=wobj0;
    MoveL PLACE6,v200,z50,Servo\WObj:=wobj0;
    Reset GripperL_7;
    MoveL PRE_PLACE6,v200,z50,Servo\WObj:=wobj0;
  ENDPROC
  PROC Path_60()
    MoveL PHOTO,v200,z50,Servo\WObj:=wobj0;
    WaitTime 5;
    MoveL PRE_TAKE,v200,z50,Servo\WObj:=wobj0;
    MoveL TAKE,v200,z50,Servo\WObj:=wobj0;
    WaitTime 1;
    Set GripperL_8;
    WaitTime 1;
    MoveL PRE_TAKE,v200,z50,Servo\WObj:=wobj0;
    MoveL PRE_PLACE7,v200,z50,Servo\WObj:=wobj0;
    MoveL PLACE7,v200,z50,Servo\WObj:=wobj0;
    Reset GripperL_8;
    MoveL PRE_PLACE7,v200,z50,Servo\WObj:=wobj0;
  ENDPROC
  PROC Path_70()
    MoveL PHOTO,v200,z50,Servo\WObj:=wobj0;
    WaitTime 5;
    MoveL PRE_TAKE,v200,z50,Servo\WObj:=wobj0;
    MoveL TAKE,v200,z50,Servo\WObj:=wobj0;
    WaitTime 1;
    Set GripperL_9;
    WaitTime 1;
    MoveL PRE_TAKE,v200,z50,Servo\WObj:=wobj0;
    MoveL PRE_PLACE8,v200,z50,Servo\WObj:=wobj0;
    MoveL PLACE8,v200,z50,Servo\WObj:=wobj0;
    Reset GripperL_9;
    MoveL PRE_PLACE8,v200,z50,Servo\WObj:=wobj0;
  ENDPROC
  PROC Path_80()
    MoveL PHOTO,v200,z50,Servo\WObj:=wobj0;
    WaitTime 5;
    MoveL PRE_TAKE,v200,z50,Servo\WObj:=wobj0;
    MoveL TAKE,v200,z50,Servo\WObj:=wobj0;
    WaitTime 1;
    Set GripperL_10;
    WaitTime 1;
    MoveL PRE_TAKE,v200,z50,Servo\WObj:=wobj0;
    MoveL PRE_PLACE9,v200,z50,Servo\WObj:=wobj0;
    MoveL PLACE9,v200,z50,Servo\WObj:=wobj0;
    Reset GripperL_10;
    MoveL PRE_PLACE9,v200,z50,Servo\WObj:=wobj0;
  ENDPROC
ENDMODULE

